Staubli VAL3: init_logAction.pgx

public program init_logAction()
  local num l_nSize
  local num i
begin
  // mutex it
  setMutex(bLogMutex)
  // logAction
  resize(sLog,1,1)
  sLog=""
  bLogMutex=false
end
